RoboDK station: Lab3_Restrepo_Penagos.rdk

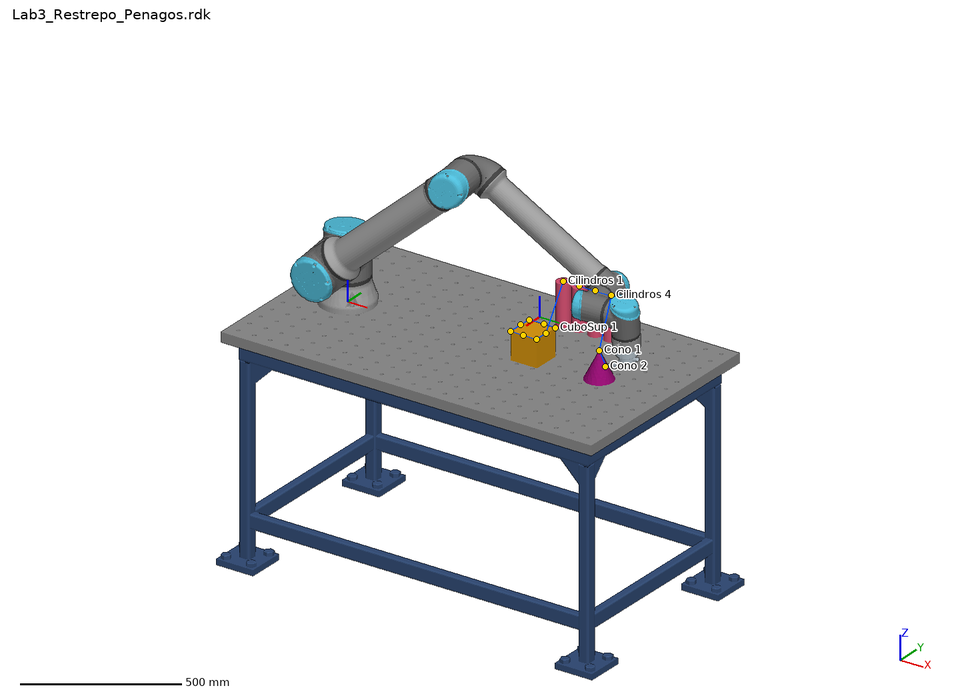
[picture v0: the station drawn from its stored meshes, robots at their saved joint values, targets as dots, program paths as lines]
Station Dispensing with UR10e #03 (saved by RoboDK 5.6.0). Poses are relative to the parent item; angles as X-Y-Z fixed-axis rotations.
Station parameters (name, value as stored): TAGS, ['Dispensing'], Palletizing Plugin
  - frame UR10e Base at (0, 0, 0) mm
    - robot UR10e: 6 axes, payload 10 kg, reach 1300 mm, repeatability 0.05 mm, weight 28.9 kg
        modified DH rows (alpha deg, a mm, theta deg, d mm): 0, 0, 0, 180.7; 90, 0, 180, 0; 0, 612.6, 0, 0; 0, 571.335, 0, 174.15; -90, 0, 0, 119.85; 90, 0, 180, 116.55
        joint limits [-360, -360, -360, -360, -360, -360] to [360, 360, 360, 360, 360, 360]; home [0, -90, -90, 0, 90, 0]; saved at [7.633, -138.909, -74.936, -58.322, 99.551, 95.323]
      - tool Generic Pencil Tool, TCP at (82, 0, 101.78) mm, rotated rx 0 ry 60 rz 0 deg, size 125 x 74.9 x 107.3 mm
    - frame Frame Dispensing at (550, 250, 0) mm, rotated rx 0 ry 0 rz -90 deg
      - object Cube 100mm at (200, 100, 0) mm, size 100 x 100 x 100 mm, geometry from Cube-100mm.sld
      - target CuboSup 1 (Cartesian target) at (200.45, 199.37, 100) mm, rotated rx -180 ry 0 rz -113.43 deg; joints [26.249, -118.879, -128.19, 25.326, 48.676, 120.507] of UR10e
      - target CuboSup 2 (Cartesian target) at (200.39, 156.5, 100) mm, rotated rx 180 ry 0 rz -113.43 deg; joints [28.205, -116.604, -133.092, 26.765, 47.23, 122.281] of UR10e
      - target CuboSup 3 (Cartesian target) at (200.76, 100.57, 100) mm, rotated rx -180 ry 0 rz -113.43 deg; joints [31.193, -113.603, -139.461, 28.142, 45.078, 125.155] of UR10e
      - target CuboSup 4 (Cartesian target) at (244.76, 100.28, 100) mm, rotated rx -180 ry 0 rz -113.43 deg; joints [26.727, -114.033, -139.847, 31.855, 48.32, 120.933] of UR10e
      - target CuboSup 5 (Cartesian target) at (299.58, 100.6, 100) mm, rotated rx -180 ry 0 rz -113.43 deg; joints [20.8, -114.681, -139.727, 35.547, 52.835, 115.956] of UR10e
      - target CuboSup 6 (Cartesian target) at (299.36, 148.16, 100) mm, rotated rx -180 ry 0 rz -113.43 deg; joints [19.003, -116.913, -134.333, 33.209, 54.241, 114.567] of UR10e
      - target CuboSup 7 (Cartesian target) at (299.6, 198.43, 100) mm, rotated rx 180 ry 0 rz -113.43 deg; joints [17.378, -119.357, -128.599, 30.619, 55.528, 113.353] of UR10e
      - target CuboSup 8 (Cartesian target) at (248.68, 199.26, 100) mm, rotated rx -180 ry 0 rz -113.43 deg; joints [22.013, -119.071, -128.553, 28.172, 51.894, 116.923] of UR10e
      - object Cylinder 50x150mm at (0, 150, 0) mm, size 50 x 50 x 150 mm, geometry from Cylinder-50x150mm.sld
      - object Cylinder 50x150mm at (0, 210, 0) mm, size 50 x 50 x 150 mm, geometry from Cylinder-50x150mm.sld
      - object Cylinder 50x150mm at (0, 90, 0) mm, size 50 x 50 x 150 mm, geometry from Cylinder-50x150mm.sld
      - object Cylinder 50x150mm at (0, 270, 0) mm, size 50 x 50 x 150 mm, geometry from Cylinder-50x150mm.sld
      - target Cilindros 1 (Cartesian target) at (0, 90, 150) mm, rotated rx -180 ry 0 rz -113.43 deg; joints [48.618, -106.408, -133.52, -1.98, 34.525, 147.062] of UR10e
      - target Cilindros 2 (Cartesian target) at (0, 150, 150) mm, rotated rx -180 ry 0 rz -113.43 deg; joints [44.405, -111.117, -127.425, 1.702, 36.674, 140.832] of UR10e
      - target Cilindros 3 (Cartesian target) at (0, 210, 150) mm, rotated rx -180 ry 0 rz -113.43 deg; joints [40.806, -115.372, -121.04, 3.383, 38.743, 136.016] of UR10e
      - target Cilindros 4 (Cartesian target) at (0, 270, 150) mm, rotated rx -180 ry 0 rz -113.43 deg; joints [37.708, -119.396, -114.386, 3.677, 40.67, 132.217] of UR10e
      - object Cone 100x100mm at (250, 400, 0) mm, size 99.5 x 100 x 100 mm, geometry from Cone-100x100mm.sld
      - target Cono 1 (Cartesian target) at (250.57, 400.61, 98.28) mm, rotated rx 135.82 ry -52.52 rz -75.79 deg; joints [3.178, -133.249, -85.137, -40.898, 112.857, 118.518] of UR10e
      - target Cono 2 (Cartesian target) at (250.91, 425.06, 49.79) mm, rotated rx 160.12 ry -61.63 rz -70.47 deg; joints [168.903, 2.456, -12.07, 104.752, 81.653, -103.6] of UR10e
    - object Table 1400x800x800mm at (140, 0, 0) mm, size 1420 x 820 x 800 mm, geometry from Table-1400x800x800mm.sld
  - program Prog1 (16 instructions, listed below)
  - program Prog2 (4 instructions, listed below)
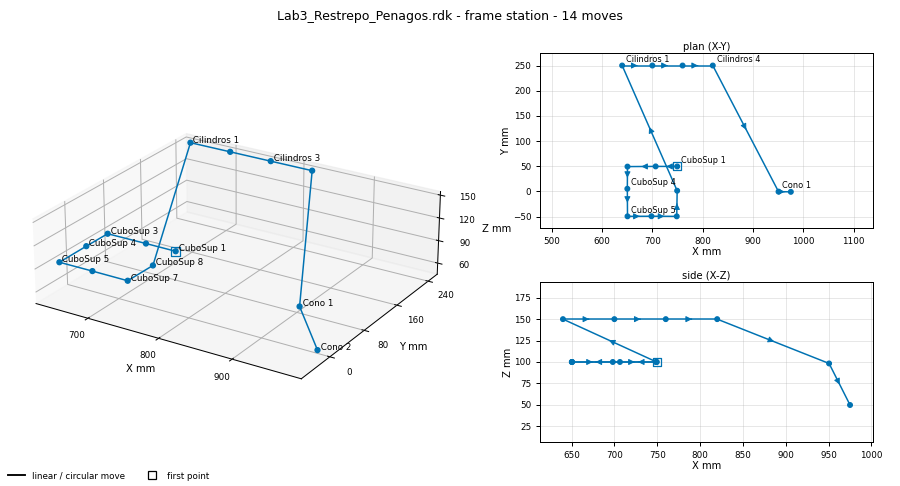
[picture p0: tool path of Lab3_Restrepo_Penagos.rdk in frame station, 14 of 16 moves have a stored position in this frame; points joined in program order, loops and branches not executed]

--- program Prog1 (robot UR10e) ---
  Set Ref.: Frame Dispensing
  Set Tool: Generic Pencil Tool
  MoveL (Target 1) -> target CuboSup 1
  MoveL (Target 2) -> target CuboSup 2
  MoveL (Target 3) -> target CuboSup 3
  MoveL (Target 4) -> target CuboSup 4
  MoveL (Target 5) -> target CuboSup 5
  MoveL (Target 6) -> target CuboSup 6
  MoveL (Target 7) -> target CuboSup 7
  MoveL (Target 8) -> target CuboSup 8
  MoveL (Cilindros 1)
  MoveL (Cilindros 2)
  MoveL (Cilindros 3)
  MoveL (Cilindros 4)
  MoveL (Cono 1)
  MoveL (Cono 2)

--- program Prog2 (robot UR10e) ---
  Set Ref.: Frame Dispensing
  Set Tool: Generic Pencil Tool
  MoveL (Cono 3) [its target is no longer in the station]
  MoveL (Cono 4) [its target is no longer in the station]
